FUNCTION_BLOCK FB_SquareWave
VAR_INPUT
	PulseLength	: DINT;		// Pulse length in [ms]
END_VAR
VAR_OUTPUT
	Value		: BOOL;
END_VAR
VAR
	Flasher_On	: TON;
	Edge		: BOOL;
END_VAR


Flasher_On(IN := NOT Flasher_On.Q, PT := DINT_TO_TIME(PulseLength));

IF Flasher_On.Q THEN
	Flasher_On(IN := FALSE);
	Edge := TRUE;
END_IF

IF Edge AND Value THEN
	Value := FALSE;
	Edge := FALSE;
ELSIF Edge AND NOT Value THEN
	Value := TRUE;
	Edge := FALSE;
END_IF

END_FUNCTION_BLOCK

(* stored: Version 1.1.0.1, ProductVersion 3.1.4022.18
   POU FB_SquareWave: Id {574db9a7-1f9a-471a-a136-1027f64c3fa0}, SpecialFunc None *)
